
// ===== library: MasterCopy "Modes" =====

FUNCTION "Modes" : Void   // FC1, LAD
TITLE = Modes Setup
{ S7_Optimized_Access := 'TRUE' }
VERSION : 0.1
BEGIN

REGION Network 1: Automatic Mode
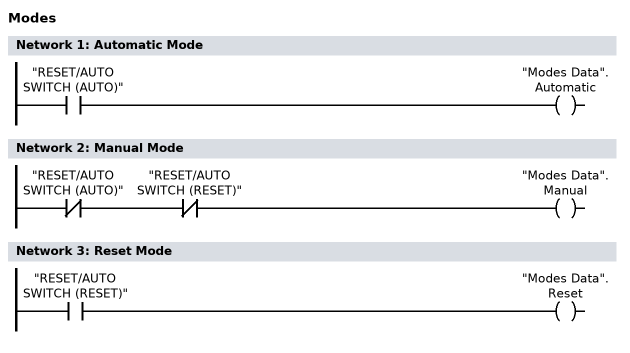
   RUNG wire#powerrail
      Contact( "RESET/AUTO SWITCH (AUTO)" )
      Coil( "Modes Data".Automatic )
   END_RUNG
   // the same network as SCL:
   "Modes Data".Automatic := "RESET/AUTO SWITCH (AUTO)";
END_REGION

REGION Network 2: Manual Mode
   RUNG wire#powerrail
      I_Contact( "RESET/AUTO SWITCH (AUTO)" )
      I_Contact( "RESET/AUTO SWITCH (RESET)" )
      Coil( "Modes Data".Manual )
   END_RUNG
   // the same network as SCL:
   "Modes Data".Manual := NOT "RESET/AUTO SWITCH (AUTO)" AND NOT "RESET/AUTO SWITCH (RESET)";
END_REGION

REGION Network 3: Reset Mode
   RUNG wire#powerrail
      Contact( "RESET/AUTO SWITCH (RESET)" )
      Coil( "Modes Data".Reset )
   END_RUNG
   // the same network as SCL:
   "Modes Data".Reset := "RESET/AUTO SWITCH (RESET)";
END_REGION

REGION Network 4: Pre-Automatic Mode
END_REGION
END_FUNCTION

// ===== library: MasterCopy "Modes Data" =====

DATA_BLOCK "Modes Data"   // DB1
{ S7_Optimized_Access := 'TRUE' }
VERSION : 0.1
   VAR
      Automatic : Bool;
      Manual : Bool;
      Reset : Bool;
      "Pre-Automatic" : Bool;
   END_VAR
BEGIN
END_DATA_BLOCK